// TIA Portal V19 export
VAR_GLOBAL   // PLC tag table "SafetyTags"
   Safety_PB_Blue_Lamp AT %M90.0 : Bool;
END_VAR
